(* CODESYS project Estacao 6 - pick and place (2022) .project

Project tree, tasks and I/O mapping:
  Device : CPX-CEC-C1-V3, Festo AG & Co. KG, order no. 3473128, version 3.5.7.37
      unmapped channels: Rotary switch
    application Application
      libraries: Standard, * (System)
      task MainTask (cyclic, interval t#20ms, priority 20) calls PLC_PRG
      program PLC_PRG [ST]
      global variables GVL
      program saida_pecas [ST]
      program pisca_pisca [ST]
      program entrada_peca [ST]
      program teste_comunicacao [ST]
    PLC_Diagnosis : PLC-Diagnosis, Festo AG & Co. KG, version 3.5.4.1
    CPX_System : CPX_System, Festo AG & Co. KG, order no. 3473128, version 1.258
      CEC_C1_V3 : CEC-C1-V3, Festo AG & Co. KG, order no. 3473128, version 1.258
          settings:  = 0;  = 228781598969344;  = 1006807232;  = 65535;  = 16885952;  = 13959208;  = 1f5d13d0;  = 5
      _8DI_8DO : 8DI/8DO, Festo AG & Co. KG, order no. 526257, version 1.258
          settings:  = 0;  = 1;  = 1;  = 1;  = 1;  = 0;  = 1;  = 1;  = 0;  = 0;  = 0;  = 0;  = 0;  = 0;  = 0;  = 0;  = 0;  = 0;  = 0;  = 0;  = 0;  = 0;  = 0;  = 0;  = 0;  = 0;  = 0;  = 0;  = 0;  = 0;  = 0;  = 0;  = 0;  = 0;  = 0;  = 0;  = 0;  = 0;  = 0;  = 0;
             = 0;  = 0;  = 0;  = 0;  = 0;  = 0;  = 0;  = 0;  = 0;  = 0;  = 0;  = 0;  = 0;  = 0;  = 0;  = 0;  = 0;  = 0;  = 0;  = 0;  = 0;  = 0;  = 0;  = 0;  = 0;  = 0;  = 0;  = 0;  = 0;  = 0;  = 0;  = 0;  = 0;  = 0;  = 0;  = 0;  = 0;  = 0;  = 0;  = 0;
             = 576751027668385792;  = 'PI%i.0.0.1=1';  = 'PI%i.0.1.1=1';  = 'PI%i.0.2.1=1';  = 'PI%i.1.0.1=1';  = 'PI%i.1.1.1=0';  = 'PI%i.1.4.2=1';  = 'PI%i.1.6.2=1';  = 'PI%i.6.0.1=0';  = 'PI%i.6.1.1=0';  = 'PI%i.6.2.1=0';  = 'PI%i.6.3.1=0';  = 'PI%i.6.4.1=0';  = 'PI%i.6.5.1=0';  = 'PI%i.6.6.1=0';  = 'PI%i.6.7.1=0';  = dd39f1de;  = 6
          unmapped channels: Input 0, Output 0
      _8DI_8DO_1 : 8DI/8DO, Festo AG & Co. KG, order no. 526257, version 1.258
          settings:  = 0;  = 1;  = 1;  = 1;  = 1;  = 0;  = 1;  = 1;  = 0;  = 0;  = 0;  = 0;  = 0;  = 0;  = 0;  = 0;  = 0;  = 0;  = 0;  = 0;  = 0;  = 0;  = 0;  = 0;  = 0;  = 0;  = 0;  = 0;  = 0;  = 0;  = 0;  = 0;  = 0;  = 0;  = 0;  = 0;  = 0;  = 0;  = 0;  = 0;
             = 0;  = 0;  = 0;  = 0;  = 0;  = 0;  = 0;  = 0;  = 0;  = 0;  = 0;  = 0;  = 0;  = 0;  = 0;  = 0;  = 0;  = 0;  = 0;  = 0;  = 0;  = 0;  = 0;  = 0;  = 0;  = 0;  = 0;  = 0;  = 0;  = 0;  = 0;  = 0;  = 0;  = 0;  = 0;  = 0;  = 0;  = 0;  = 0;  = 0;
             = 576751027668385792;  = 'PI%i.0.0.1=1';  = 'PI%i.0.1.1=1';  = 'PI%i.0.2.1=1';  = 'PI%i.1.0.1=1';  = 'PI%i.1.1.1=0';  = 'PI%i.1.4.2=1';  = 'PI%i.1.6.2=1';  = 'PI%i.6.0.1=0';  = 'PI%i.6.1.1=0';  = 'PI%i.6.2.1=0';  = 'PI%i.6.3.1=0';  = 'PI%i.6.4.1=0';  = 'PI%i.6.5.1=0';  = 'PI%i.6.6.1=0';  = 'PI%i.6.7.1=0';  = dd307755;  = 6
          unmapped channels: Input 0, Output 0
    Ethernet : Ethernet, 3S - Smart Software Solutions GmbH, version 3.5.10.0
        settings: IPAddress = [192,168,2,60]; SubnetMask = [255,255,0,0]; GatewayAddress = [192,168,1,1]; MACAddress = [16#00,16#0E,16#F0,16#5D,16#13,16#D0]; NetworkInterfaceName = 'eth0'; NetworkInterfaceName = "eth0"; SaveCommunicationSettings = FALSE
      ModbusTCP_Slave_Device : ModbusTCP Slave Device, 3S - Smart Software Solutions GmbH, version 3.5.10.0
          unmapped channels: Inputs, Outputs
*)

// Device/Application/GVL
{attribute 'qualified_only'}
VAR_GLOBAL
//Entradas
//Sensores
	S_meio 			AT %IX1.0 :BOOL; //Sesnor do inicio da esteira
	S_inicio 	 	AT %IX1.1 :BOOL; //Sensor do meio da esteira
	S_fim			AT %IX1.2 :BOOL; //Sensor do fim da esteira
	//			AT %IX1.3 :BOOL;
	Mani_recuado 	AT %IX1.4  :BOOL; //Manipulaor recuado
	Mani_Avancado 	AT %IX1.5  :BOOL; //Manipulador avancado
	Mani_Superior	AT %IX1.6  :BOOL; //Manipulador na posição superior
	Peca_sugada 	AT %IX1.7  :BOOL; //Peça sugada pela ventosa
	
//IHM
	Start_btn 		AT	%IX2.0	:BOOL;  //Botão de start
	Stop_btn 		AT	%IX2.1	:BOOL;	//Botão de stop (NF)
	Chave 			AT	%IX2.2	:BOOL;	//Chave auto/manual
	Reset_btn 		AT	%IX2.3	:BOOL;	//Botão de reset
	I4_IHM			AT	%IX2.4	:BOOL;	//Bit de entrada 4 da IHM
	I5_IHM			AT	%IX2.5	:BOOL;	//Bit de entrada 5 da IHM
	I6_IHM 			AT	%IX2.6	:BOOL;	//Bit de entrada 6 da IHM
	I7_IHM			AT	%IX2.7	:BOOL;	//Bit de entrada 7 da IHM

	
//Saídas

	E_Entrando 	AT	%QX0.1	:BOOL;	//Esteira no sentido de entrada de peças
	E_saindo 	AT	%QX0.0	:BOOL;	//Esteira no sentido de saída de peças
	Separador 	AT	%QX0.2	:BOOL;	//Ativar o separador
	Recuar_mani	AT	%QX0.4	:BOOL;	//
	Avanca_mani AT	%QX0.5	:BOOL;	//
	Descer_mani AT	%QX0.6	:BOOL;	//
	Ativar_vac	AT	%QX0.7	:BOOL;	//
		

//IHM				
	Start_LED		AT	%QX1.0	:BOOL;	//LED do botão de start
	Reset_LED 		AT	%QX1.1	:BOOL;	//LED do botão de reset
	Q1_LED 			AT	%QX1.2	:BOOL;	//LED sinalizador Q1
	Q2_LED			AT	%QX1.3	:BOOL;	//LED sinalizador Q2
	Q4_IHM			AT	%QX1.5	:BOOL;	//Saída Q4 IHM 
	Q5_IHM			AT	%QX1.4	:BOOL;	//Saída Q5 IHM 
	Q6_IHM			AT	%QX1.6	:BOOL;	//Saída Q6 IHM
	Q7_IHM 			AT	%QX1.7	:BOOL;	//Saída Q7 IHM
	
	
	flag_btn_visu :BOOL;
	btn_armazena :  BOOL;
	
	modo_entrada: BOOL := FALSE;
	modo_saida: BOOL := FALSE;
	ligar_pisca: BOOL := FALSE;
	
	estacao_processo : BOOL;
	estacao_iniciada : BOOL;
	parada_geral : BOOL := FALSE;
	reset_geral : BOOL := FALSE;
	
	estacao_em_processo : BOOL;
	
	flag_modo_saida : BOOL :=	FALSE; // Flag utilizada na hora da liberação de peças pela estação 7
	
	//MODBUS bits
	//Entradas
	Mod_I_0_0 		AT %IX4.0 : BOOL;//start
	Mod_I_0_1	 	AT %IX4.1 : BOOL;//stop
	Mod_I_0_2 		AT %IX4.2 : BOOL;//reset
	Mod_I_0_3 		AT %IX4.3 : BOOL;//Modo entrada
	Mod_I_0_4 		AT %IX4.4 : BOOL;//Teste de resposta da estação - IN	
	Mod_I_0_5 		AT %IX4.5 : BOOL;//
	Mod_I_0_6 		AT %IX4.6 : BOOL;//
	Mod_I_0_7 		AT %IX4.7 : BOOL;//
	
	//Saídas
	Mod_Q_0_0 		AT %QX2.0 : BOOL; //Estação iniciada 
	Mod_Q_0_1	 	AT %QX2.1 : BOOL; //Estação parada 		
	Mod_Q_0_2 		AT %QX2.2 : BOOL; //Estação em processo			
	Mod_Q_0_3 		AT %QX2.3 : BOOL; //Estação em modo de entrada
	Mod_Q_0_4 		AT %QX2.4 : BOOL; //Estação em modo de saída
	Mod_Q_0_5 		AT %QX2.5 : BOOL; //Teste de resposta da estação - OUT
	Mod_Q_0_6 		AT %QX2.6 : BOOL;
	Mod_Q_0_7 		AT %QX2.7 : BOOL; 
	
	
	
	
END_VAR

// Device/Application/PLC_PRG
PROGRAM PLC_PRG
VAR
	x : bool;
END_VAR

teste_comunicacao();

gvl.Mod_Q_0_0 := gvl.estacao_iniciada;
gvl.Mod_Q_0_1 := gvl.parada_geral;
gvl.Mod_Q_0_2 := gvl.estacao_processo;
gvl.Mod_Q_0_3 := gvl.modo_entrada;
gvl.Mod_Q_0_4 := gvl.modo_saida;




IF NOT gvl.parada_geral AND gvl.estacao_iniciada THEN
	gvl.Q1_LED := TRUE;
	entrada_peca();
	saida_pecas();
	pisca_pisca();	
END_IF	

IF  gvl.parada_geral THEN 
	gvl.Q1_LED := FALSE;
	gvl.E_Entrando := FALSE;
	gvl.E_saindo := FALSE;
	gvl.modo_entrada := FALSE; 
	gvl.modo_saida := FALSE;
	gvl.ligar_pisca := FALSE;
END_IF

IF gvl.reset_geral THEN
	gvl.Separador := FALSE;
	gvl.parada_geral := FALSE;
	gvl.reset_geral := FALSE;
END_IF

IF gvl.Mod_I_0_3 AND NOT gvl.Mod_I_0_4 THEN
	gvl.modo_entrada := TRUE; 
	gvl.modo_saida := FALSE;
END_IF

IF NOT gvl.Mod_I_0_3 AND gvl.Mod_I_0_4 THEN
	gvl.modo_saida := TRUE; 
	gvl.modo_entrada := FALSE; 
END_IF

IF gvl.Mod_I_0_0 OR gvl.Start_btn THEN
	IF NOT gvl.parada_geral THEN
		gvl.estacao_iniciada := TRUE;	
	END_IF
END_IF


IF gvl.Mod_I_0_1 OR NOT gvl.Stop_btn THEN
	gvl.estacao_iniciada := FALSE;
	gvl.parada_geral := TRUE;
END_IF

IF gvl.Mod_I_0_2 OR gvl.Reset_btn THEN
	gvl.reset_geral := TRUE;
END_IF

END_PROGRAM

// Device/Application/teste_comunicacao
PROGRAM teste_comunicacao
VAR
	
	TON_temp_1: TON;
	TON_1: BOOL;	

END_VAR

gvl.Mod_Q_0_5 := gvl.Mod_I_0_5;

END_PROGRAM

// Device/Application/entrada_peca
PROGRAM entrada_peca
VAR
	PASSOS :INT;

	TON_temp_1: TON;
	TON_1: BOOL;
	
	TON_temp_2: TON;
	TON_2: BOOL;
	
	TON_temp_3: TON;
	TON_3: BOOL;
	
	TON_temp_4: TON;
	TON_4: BOOL;
	
	finalizou : BOOL;
	primeira_peca : BOOL;
	flag_peca_disponibilizada : BOOL;

END_VAR

TON_temp_1(IN := TON_1, PT:= T#1S);
TON_temp_2(IN := TON_2, PT:= T#6S);
TON_temp_3(IN := TON_3, PT:= T#2.5S);
TON_temp_4(IN := TON_4, PT:= T#0.5S);

IF gvl.modo_entrada AND NOT gvl.modo_saida THEN //Caso o modo entrada seja ativado e o saída dessativado
	
	IF gvl.S_inicio THEN
		gvl.E_Entrando := TRUE;
		gvl.E_Entrando := TRUE;
		gvl.ligar_pisca := TRUE;
		gvl.estacao_processo := TRUE; 
		gvl.estacao_em_processo := TRUE;
		IF NOT primeira_peca THEN
			primeira_peca := TRUE;
			gvl.Separador := TRUE;
		END_IF
	END_IF
	
	IF TON_temp_4.Q THEN
		TON_4 := FALSE;
		gvl.Separador  := FALSE;
	END_IF
	
	IF gvl.S_meio AND gvl.I4_IHM THEN
		flag_peca_disponibilizada := TRUE;
		TON_4 := TRUE;
		
		gvl.E_Entrando := TRUE;
	END_IF
	
	IF NOT gvl.S_fim AND flag_peca_disponibilizada THEN
		flag_peca_disponibilizada := FALSE;
		TON_1 := TRUE;
	END_IF
	
	IF TON_temp_1.Q THEN
		TON_1 := FALSE;
		TON_3 := TRUE;
		gvl.Separador := TRUE;
	END_IF
	
	IF TON_temp_3.q AND NOT gvl.S_inicio AND NOT gvl.S_inicio THEN
		gvl.E_Entrando := FALSE;
		TON_3 := FALSE;
	END_IF
	
	IF gvl.S_meio AND NOT gvl.S_inicio AND NOT gvl.I4_IHM AND NOT TON_3  AND NOT TON_1 THEN //
		gvl.E_Entrando := FALSE;
	END_IF
	
	IF NOT gvl.S_inicio AND NOT gvl.S_meio AND gvl.S_fim AND gvl.I4_IHM THEN
		TON_2 := TRUE;
	ELSE
		TON_2 := FALSE;
	END_IF
	
	IF TON_temp_2.Q THEN
		gvl.E_Entrando := FALSE; //Desliga a esteira
		gvl.Separador := FALSE; //Desliga o separador
		primeira_peca := FALSE;
		gvl.estacao_em_processo := false;
		//gvl.modo_entrada := FALSE;
		gvl.ligar_pisca := FALSE; //Desliga o pisca pisca
		gvl.estacao_processo := FALSE; 
		TON_2 := FALSE;
	END_IF

END_IF

END_PROGRAM

// Device/Application/saida_pecas
PROGRAM saida_pecas
VAR
	
	TON_temp_esteira: TON;
	TON_esteira: BOOL;	
	
	TON_temp_1: TON;
	TON_1: BOOL;	

END_VAR

TON_temp_esteira(IN := TON_esteira, PT:= T#3S);
TON_temp_1(IN := TON_1, PT:= T#1S);

IF gvl.modo_saida THEN
	
	//Sinal da estação 7 sinalizando uma peça disponível
	IF gvl.I4_IHM THEN
		TON_1 := TRUE;
	END_IF
	
	
	IF TON_temp_1.Q AND NOT gvl.I4_IHM and not gvl.S_fim THEN
		TON_1 := FALSE;
		gvl.flag_modo_saida := TRUE;
	END_IF	
	////////////////////////////////////////////////////

	IF gvl.flag_modo_saida THEN
		gvl.flag_modo_saida := FALSE;
		gvl.estacao_em_processo:= TRUE;
		gvl.ligar_pisca := TRUE;
		gvl.estacao_processo := TRUE; 
		gvl.E_saindo := TRUE;
		gvl.Separador := FALSE;	
	END_IF
	
	IF gvl.S_inicio  THEN
		TON_esteira := TRUE;
	END_IF
	 
	IF TON_temp_esteira.Q THEN
		TON_esteira := FALSE;
		gvl.ligar_pisca := FALSE;
		gvl.estacao_processo := FALSE; 
		gvl.E_saindo := FALSE;
		gvl.estacao_em_processo := false;
		//gvl.flag_modo_saida := FALSE;
	END_IF


END_IF

END_PROGRAM

// Device/Application/pisca_pisca
PROGRAM pisca_pisca
VAR
	
	TON_temp_1: TON;
	TON_1: BOOL;
	TON_temp_2: TON;
	TON_2: BOOL;
	
	passo: INT;
END_VAR

TON_temp_1(IN := TON_1, PT:= T#0.2S);
TON_temp_2(IN := TON_2, PT:= T#0.2S);


IF gvl.ligar_pisca AND (passo = 0)  THEN
	TON_1 := TRUE;
	passo := 1;
END_IF


IF NOT gvl.ligar_pisca THEN
	TON_1 := FALSE;
	TON_2 := FALSE;
	GVL.Q2_LED := FALSE;
	passo := 0;
END_IF

IF TON_temp_1.Q THEN
	TON_1 := FALSE;
	TON_2 := TRUE;
	GVL.Q2_LED := TRUE;
END_IF
IF TON_temp_2.Q THEN
	TON_1 := TRUE;
	TON_2 := FALSE;
	GVL.Q2_LED := FALSE;
END_IF

END_PROGRAM
